// TIA Portal V19 export
TYPE "LEXCHANGETRAY_typeHandlingXyzEm_interface"
// stored: Access Published
   STRUCT
      deliver : "LEXCHANGETRAY_typeHandlingXyzEm_deliver_interface";
      recieve : "LEXCHANGETRAY_typeHandlingXyzEm_recieve_interface";
   END_STRUCT;
END_TYPE
